// TIA Portal V21 export
DATA_BLOCK "ConfigDB"   // DB3
{ S7_Optimized_Access := 'TRUE' }
// stored: MemoryReserve 100
   VAR
      ksd1 : "coneCrusherConfigs";
   END_VAR
BEGIN
   ksd1.luS.self.timeToEstablishReturnFlow := T#60s;
   ksd1.luS.self.timeToEstablishFlow := T#15s;
   ksd1.luS.self.minOilFlow := 110.0;
   ksd1.luS.localModeSwitch.referenceDesignator := WSTRING#'LusLocalModeSw';
   ksd1.luS.localModeSwitch.onDelay := T#500ms;
   ksd1.luS.localModeSwitch.offDelay := T#200ms;
   ksd1.luS.btnStart.referenceDesignator := WSTRING#'LusBtnStart';
   ksd1.luS.btnStart.onDelay := T#500ms;
   ksd1.luS.btnStart.offDelay := T#200ms;
   ksd1.luS.btnStop.referenceDesignator := WSTRING#'LusBtnStop';
   ksd1.luS.btnStop.onDelay := T#500ms;
   ksd1.luS.btnStop.offDelay := T#200ms;
   ksd1.luS.btnReset.referenceDesignator := WSTRING#'LusBtnReset';
   ksd1.luS.btnReset.onDelay := T#500ms;
   ksd1.luS.btnReset.offDelay := T#200ms;
   ksd1.luS.oilPump1SelSwitch.referenceDesignator := WSTRING#'OilPump1Selected';
   ksd1.luS.oilPump1SelSwitch.onDelay := T#500ms;
   ksd1.luS.oilPump1SelSwitch.offDelay := T#200ms;
   ksd1.luS.oilPump2SelSwitch.referenceDesignator := WSTRING#'OilPump2Selected';
   ksd1.luS.oilPump2SelSwitch.onDelay := T#500ms;
   ksd1.luS.oilPump2SelSwitch.offDelay := T#200ms;
   ksd1.luS.oilPreparationSwitch.referenceDesignator := WSTRING#'OilPreparationSw';
   ksd1.luS.oilPreparationSwitch.onDelay := T#500ms;
   ksd1.luS.oilPreparationSwitch.offDelay := T#200ms;
   ksd1.luS.returnOilFlowSwitch.referenceDesignator := WSTRING#'ReturnOilFlowSw';
   ksd1.luS.returnOilFlowSwitch.onDelay := T#500ms;
   ksd1.luS.returnOilFlowSwitch.offDelay := T#200ms;
   ksd1.luS.oilLevelMax.referenceDesignator := WSTRING#'OilLevelMax';
   ksd1.luS.oilLevelMax.onDelay := T#500ms;
   ksd1.luS.oilLevelMax.offDelay := T#200ms;
   ksd1.luS.oilLevelMid.referenceDesignator := WSTRING#'OilLevelMid';
   ksd1.luS.oilLevelMid.onDelay := T#500ms;
   ksd1.luS.oilLevelMid.offDelay := T#200ms;
   ksd1.luS.oilLevelMin.referenceDesignator := WSTRING#'OilLevelMin';
   ksd1.luS.oilLevelMin.onDelay := T#500ms;
   ksd1.luS.oilLevelMin.offDelay := T#200ms;
   ksd1.luS.oilTempSwitchHigh.referenceDesignator := WSTRING#'OilTempSwHigh';
   ksd1.luS.oilTempSwitchHigh.onDelay := T#500ms;
   ksd1.luS.oilTempSwitchHigh.offDelay := T#200ms;
   ksd1.luS.oilTempSwitchLow.referenceDesignator := WSTRING#'OilTempSwLow';
   ksd1.luS.oilTempSwitchLow.onDelay := T#500ms;
   ksd1.luS.oilTempSwitchLow.offDelay := T#200ms;
   ksd1.luS.fbPump1.referenceDesignator := WSTRING#'FbPump1';
   ksd1.luS.fbPump1.onDelay := T#500ms;
   ksd1.luS.fbPump1.offDelay := T#200ms;
   ksd1.luS.fbPump2.referenceDesignator := WSTRING#'FbPump2';
   ksd1.luS.fbPump2.onDelay := T#500ms;
   ksd1.luS.fbPump2.offDelay := T#200ms;
   ksd1.luS.pump1Fault.referenceDesignator := WSTRING#'Pump1Fault';
   ksd1.luS.pump1Fault.onDelay := T#500ms;
   ksd1.luS.pump1Fault.offDelay := T#200ms;
   ksd1.luS.pump2Fault.referenceDesignator := WSTRING#'Pump2Fault';
   ksd1.luS.pump2Fault.onDelay := T#500ms;
   ksd1.luS.pump2Fault.offDelay := T#200ms;
   ksd1.luS.oilTempTank.referenceDesignator := WSTRING#'OilTempTank';
   ksd1.luS.oilTempTank.physicalUnit := 'C';
   ksd1.luS.oilTempTank.limitHigh2 := 60.0;
   ksd1.luS.oilTempTank.limitHigh1 := 55.0;
   ksd1.luS.oilTempTank.processValueMax := 120.0;
   ksd1.luS.oilTempTank.processValueMin := -50.0;
   ksd1.luS.oilTempTank.scaleAnalogUppPoint := 27648.0;
   ksd1.luS.oilTempTank.scaleProcessUppPoint := 120.0;
   ksd1.luS.oilTempTank.scaleProcessLowPoint := -50.0;
   ksd1.luS.oilPump1.referenceDesignator := WSTRING#'Pump1';
   ksd1.luS.oilPump1.startingControlTime := T#3s;
   ksd1.luS.oilPump1.stoppingControlTime := T#2s;
   ksd1.luS.oilPump1.disableFeedbackRunning := FALSE;
   ksd1.luS.oilPump1.disableFeedbackError := FALSE;
   ksd1.luS.oilPump2.referenceDesignator := WSTRING#'OilPump2';
   ksd1.luS.oilPump2.startingControlTime := T#3s;
   ksd1.luS.oilPump2.stoppingControlTime := T#2s;
   ksd1.luS.oilPump2.disableFeedbackRunning := FALSE;
   ksd1.luS.oilPump2.disableFeedbackError := FALSE;
   ksd1.luS.returnOilTemp.referenceDesignator := WSTRING#'ReturnOilTemp';
   ksd1.luS.returnOilTemp.physicalUnit := 'C';
   ksd1.luS.returnOilTemp.isUnipolarSignal := TRUE;
   ksd1.luS.returnOilTemp.limitHigh2 := 63.0;
   ksd1.luS.returnOilTemp.limitHigh1 := 60.0;
   ksd1.luS.returnOilTemp.processValueMax := 120.0;
   ksd1.luS.returnOilTemp.processValueMin := -50.0;
   ksd1.luS.returnOilTemp.scaleAnalogUppPoint := 27648.0;
   ksd1.luS.returnOilTemp.scaleAnalogLowPoint := 0.0;
   ksd1.luS.returnOilTemp.scaleProcessUppPoint := 120.0;
   ksd1.luS.returnOilTemp.scaleProcessLowPoint := -50.0;
   ksd1.luS.oilFlow.referenceDesignator := WSTRING#'OilFlow';
   ksd1.luS.oilFlow.physicalUnit := 'l/m';
   ksd1.luS.oilFlow.limitHigh2 := 500.0;
   ksd1.luS.oilFlow.limitHigh1 := 300.0;
   ksd1.luS.oilFlow.limitLow1 := 120.0;
   ksd1.luS.oilFlow.limitLow2 := 110.0;
   ksd1.luS.oilFlow.processValueMax := 300.0;
   ksd1.luS.oilFlow.processValueMin := 0.0;
   ksd1.luS.oilFlow.scaleAnalogUppPoint := 27648.0;
   ksd1.luS.oilFlow.scaleProcessUppPoint := 300.0;
   ksd1.luS.oilFlow.scaleProcessLowPoint := 0.0;
   ksd1.luS.inletWaterTemperature.referenceDesignator := WSTRING#'InletWaterTemp';
   ksd1.luS.inletWaterTemperature.physicalUnit := 'C';
   ksd1.luS.inletWaterTemperature.processValueMax := 120.0;
   ksd1.luS.inletWaterTemperature.processValueMin := -50.0;
   ksd1.luS.inletWaterTemperature.scaleAnalogUppPoint := 27648.0;
   ksd1.luS.inletWaterTemperature.scaleProcessUppPoint := 120.0;
   ksd1.luS.inletWaterTemperature.scaleProcessLowPoint := -50.0;
   ksd1.luS.outletWaterTemperature.referenceDesignator := WSTRING#'OutletWatertemp';
   ksd1.luS.outletWaterTemperature.physicalUnit := 'C';
   ksd1.luS.outletWaterTemperature.processValueMax := 120.0;
   ksd1.luS.outletWaterTemperature.processValueMin := -50.0;
   ksd1.luS.outletWaterTemperature.scaleAnalogUppPoint := 27648.0;
   ksd1.luS.outletWaterTemperature.scaleProcessUppPoint := 120.0;
   ksd1.luS.outletWaterTemperature.scaleProcessLowPoint := -50.0;
   ksd1.luS.inletOilTemperature.referenceDesignator := WSTRING#'InletOilTemp';
   ksd1.luS.inletOilTemperature.physicalUnit := 'C';
   ksd1.luS.inletOilTemperature.processValueMax := 120.0;
   ksd1.luS.inletOilTemperature.processValueMin := -50.0;
   ksd1.luS.inletOilTemperature.scaleAnalogUppPoint := 27648.0;
   ksd1.luS.inletOilTemperature.scaleAnalogLowPoint := 0.0;
   ksd1.luS.inletOilTemperature.scaleProcessUppPoint := 120.0;
   ksd1.luS.inletOilTemperature.scaleProcessLowPoint := -50.0;
   ksd1.luS.inletOilPressure.referenceDesignator := WSTRING#'InletOilPressure';
   ksd1.luS.inletOilPressure.physicalUnit := 'bar';
   ksd1.luS.inletOilPressure.processValueMax := 16.0;
   ksd1.luS.inletOilPressure.processValueMin := 0.0;
   ksd1.luS.inletOilPressure.scaleAnalogUppPoint := 27648.0;
   ksd1.luS.inletOilPressure.scaleAnalogLowPoint := 0.0;
   ksd1.luS.inletOilPressure.scaleProcessUppPoint := 16.0;
   ksd1.luS.inletOilPressure.scaleProcessLowPoint := 0.0;
   ksd1.luS.pump1Start.referenceDesignator := WSTRING#'Pump1Start';
   ksd1.luS.pump2Start.referenceDesignator := WSTRING#'Pump2Start';
   ksd1.luS.heaterOn.referenceDesignator := WSTRING#'HeaterOn';
   ksd1.luS.waterVlvOpen.referenceDesignator := WSTRING#'WaterVlvOpen';
   ksd1.luS.oilToCoolerVlv.referenceDesignator := WSTRING#'OilToCoolerVlv';
   ksd1.btnStart.referenceDesignator := WSTRING#'CrusherBtnStart';
   ksd1.btnStart.onDelay := T#500ms;
   ksd1.btnStart.offDelay := T#200ms;
   ksd1.btnStop.referenceDesignator := WSTRING#'CrusherBtnStop';
   ksd1.btnStop.onDelay := T#500ms;
   ksd1.btnStop.offDelay := T#200ms;
   ksd1.keySwitch.referenceDesignator := WSTRING#'CrusherKeySwitch';
   ksd1.keySwitch.onDelay := T#500ms;
   ksd1.emStop.referenceDesignator := WSTRING#'EmergencyStop';
   ksd1.emStop.onDelay := T#500ms;
   ksd1.btnReset.referenceDesignator := WSTRING#'CrusherBtnReset';
   ksd1.btnReset.onDelay := T#500ms;
   ksd1.btnReset.offDelay := T#200ms;
   ksd1.btnStartLuS.referenceDesignator := WSTRING#'CrusherBtnStartLus';
   ksd1.btnStartLuS.onDelay := T#500ms;
   ksd1.btnStartLuS.offDelay := T#200ms;
   ksd1.btnStopLuS.referenceDesignator := WSTRING#'CrusherBtnStopLus';
   ksd1.btnStopLuS.onDelay := T#500ms;
   ksd1.btnStopLuS.offDelay := T#200ms;
   ksd1.premoldingSw.referenceDesignator := WSTRING#'PremoldingSw';
   ksd1.premoldingSw.onDelay := T#500ms;
   ksd1.premoldingSw.offDelay := T#500ms;
   ksd1.crusherEccentricTemp.referenceDesignator := WSTRING#'EccentricTemp';
   ksd1.crusherEccentricTemp.physicalUnit := 'C';
   ksd1.crusherEccentricTemp.isUnipolarSignal := TRUE;
   ksd1.crusherEccentricTemp.limitHigh2 := 70.0;
   ksd1.crusherEccentricTemp.limitHigh1 := 60.0;
   ksd1.crusherEccentricTemp.processValueMax := 120.0;
   ksd1.crusherEccentricTemp.processValueMin := -50.0;
   ksd1.crusherEccentricTemp.scaleAnalogUppPoint := 27648.0;
   ksd1.crusherEccentricTemp.scaleAnalogLowPoint := 0.0;
   ksd1.crusherEccentricTemp.scaleProcessUppPoint := 120.0;
   ksd1.crusherEccentricTemp.scaleProcessLowPoint := -50.0;
   ksd1.crusherOuterBearingTemp.referenceDesignator := WSTRING#'CrusherOuterBearTemp';
   ksd1.crusherOuterBearingTemp.physicalUnit := 'C';
   ksd1.crusherOuterBearingTemp.isUnipolarSignal := TRUE;
   ksd1.crusherOuterBearingTemp.limitHigh2 := 70.0;
   ksd1.crusherOuterBearingTemp.limitHigh1 := 60.0;
   ksd1.crusherOuterBearingTemp.processValueMax := 120.0;
   ksd1.crusherOuterBearingTemp.processValueMin := -50.0;
   ksd1.crusherOuterBearingTemp.scaleAnalogUppPoint := 27648.0;
   ksd1.crusherOuterBearingTemp.scaleAnalogLowPoint := 0.0;
   ksd1.crusherOuterBearingTemp.scaleProcessUppPoint := 120.0;
   ksd1.crusherOuterBearingTemp.scaleProcessLowPoint := -50.0;
   ksd1.crusherInnerBearingTemp.referenceDesignator := WSTRING#'CrusherInnerBearTemp';
   ksd1.crusherInnerBearingTemp.physicalUnit := 'C';
   ksd1.crusherInnerBearingTemp.isUnipolarSignal := TRUE;
   ksd1.crusherInnerBearingTemp.limitHigh2 := 70.0;
   ksd1.crusherInnerBearingTemp.limitHigh1 := 60.0;
   ksd1.crusherInnerBearingTemp.processValueMax := 120.0;
   ksd1.crusherInnerBearingTemp.processValueMin := -50.0;
   ksd1.crusherInnerBearingTemp.scaleAnalogUppPoint := 27648.0;
   ksd1.crusherInnerBearingTemp.scaleAnalogLowPoint := 0.0;
   ksd1.crusherInnerBearingTemp.scaleProcessUppPoint := 120.0;
   ksd1.crusherInnerBearingTemp.scaleProcessLowPoint := -50.0;
   ksd1.driveFrontBearingTemp.referenceDesignator := WSTRING#'DriveFrontBearTemp';
   ksd1.driveFrontBearingTemp.physicalUnit := 'C';
   ksd1.driveFrontBearingTemp.isUnipolarSignal := TRUE;
   ksd1.driveFrontBearingTemp.limitHigh2 := 70.0;
   ksd1.driveFrontBearingTemp.limitHigh1 := 60.0;
   ksd1.driveFrontBearingTemp.processValueMax := 120.0;
   ksd1.driveFrontBearingTemp.processValueMin := -50.0;
   ksd1.driveFrontBearingTemp.scaleAnalogUppPoint := 27648.0;
   ksd1.driveFrontBearingTemp.scaleAnalogLowPoint := 0.0;
   ksd1.driveFrontBearingTemp.scaleProcessUppPoint := 120.0;
   ksd1.driveFrontBearingTemp.scaleProcessLowPoint := -50.0;
   ksd1.driveRearBearingTemp.referenceDesignator := WSTRING#'DriveRearBearTemp';
   ksd1.driveRearBearingTemp.physicalUnit := 'C';
   ksd1.driveRearBearingTemp.isUnipolarSignal := TRUE;
   ksd1.driveRearBearingTemp.limitHigh2 := 70.0;
   ksd1.driveRearBearingTemp.limitHigh1 := 60.0;
   ksd1.driveRearBearingTemp.processValueMax := 120.0;
   ksd1.driveRearBearingTemp.processValueMin := -50.0;
   ksd1.driveRearBearingTemp.scaleAnalogUppPoint := 27648.0;
   ksd1.driveRearBearingTemp.scaleAnalogLowPoint := 0.0;
   ksd1.driveRearBearingTemp.scaleProcessUppPoint := 120.0;
   ksd1.driveRearBearingTemp.scaleProcessLowPoint := -50.0;
   ksd1.driveWindingTempP1.referenceDesignator := WSTRING#'DriveWindingTempP1';
   ksd1.driveWindingTempP1.physicalUnit := 'C';
   ksd1.driveWindingTempP1.isUnipolarSignal := TRUE;
   ksd1.driveWindingTempP1.default := 0.0;
   ksd1.driveWindingTempP1.limitHigh2 := 80.0;
   ksd1.driveWindingTempP1.limitHigh1 := 70.0;
   ksd1.driveWindingTempP1.limitLow1 := -200.0;
   ksd1.driveWindingTempP1.limitLow2 := -270.0;
   ksd1.driveWindingTempP1.processValueMax := 120.0;
   ksd1.driveWindingTempP1.processValueMin := -50.0;
   ksd1.driveWindingTempP1.scaleAnalogUppPoint := 27648.0;
   ksd1.driveWindingTempP1.scaleAnalogLowPoint := 0.0;
   ksd1.driveWindingTempP1.scaleProcessUppPoint := 120.0;
   ksd1.driveWindingTempP1.scaleProcessLowPoint := -50.0;
   ksd1.driveWindingTempP1.disableAlarms := FALSE;
   ksd1.driveWindingTempP2.referenceDesignator := WSTRING#'DriveWindingTempP2';
   ksd1.driveWindingTempP2.physicalUnit := 'C';
   ksd1.driveWindingTempP2.isUnipolarSignal := TRUE;
   ksd1.driveWindingTempP2.default := 0.0;
   ksd1.driveWindingTempP2.limitHigh2 := 80.0;
   ksd1.driveWindingTempP2.limitHigh1 := 70.0;
   ksd1.driveWindingTempP2.limitLow1 := -200.0;
   ksd1.driveWindingTempP2.limitLow2 := -270.0;
   ksd1.driveWindingTempP2.processValueMax := 120.0;
   ksd1.driveWindingTempP2.processValueMin := -50.0;
   ksd1.driveWindingTempP2.scaleAnalogUppPoint := 27648.0;
   ksd1.driveWindingTempP2.scaleAnalogLowPoint := 0.0;
   ksd1.driveWindingTempP2.scaleProcessUppPoint := 120.0;
   ksd1.driveWindingTempP2.scaleProcessLowPoint := -50.0;
   ksd1.driveWindingTempP2.disableAlarms := FALSE;
   ksd1.driveWindingTempP3.referenceDesignator := WSTRING#'DriveWindingTempP3';
   ksd1.driveWindingTempP3.physicalUnit := 'C';
   ksd1.driveWindingTempP3.isUnipolarSignal := TRUE;
   ksd1.driveWindingTempP3.default := 0.0;
   ksd1.driveWindingTempP3.limitHigh2 := 80.0;
   ksd1.driveWindingTempP3.limitHigh1 := 70.0;
   ksd1.driveWindingTempP3.limitLow1 := -200.0;
   ksd1.driveWindingTempP3.limitLow2 := -270.0;
   ksd1.driveWindingTempP3.processValueMax := 120.0;
   ksd1.driveWindingTempP3.processValueMin := -50.0;
   ksd1.driveWindingTempP3.scaleAnalogUppPoint := 27648.0;
   ksd1.driveWindingTempP3.scaleAnalogLowPoint := 0.0;
   ksd1.driveWindingTempP3.scaleProcessUppPoint := 120.0;
   ksd1.driveWindingTempP3.scaleProcessLowPoint := -50.0;
   ksd1.driveWindingTempP3.disableAlarms := FALSE;
   ksd1.driveCurrent.referenceDesignator := WSTRING#'DriveCurrent';
   ksd1.driveCurrent.physicalUnit := 'A';
   ksd1.driveCurrent.isUnipolarSignal := TRUE;
   ksd1.driveCurrent.default := 0.0;
   ksd1.driveCurrent.limitHigh2 := 100.0;
   ksd1.driveCurrent.limitHigh1 := 80.0;
   ksd1.driveCurrent.limitLow1 := -200.0;
   ksd1.driveCurrent.limitLow2 := -270.0;
   ksd1.driveCurrent.processValueMax := 200.0;
   ksd1.driveCurrent.processValueMin := 0.0;
   ksd1.driveCurrent.scaleAnalogUppPoint := 27648.0;
   ksd1.driveCurrent.scaleAnalogLowPoint := 0.0;
   ksd1.driveCurrent.scaleProcessUppPoint := 200.0;
   ksd1.driveCurrent.scaleProcessLowPoint := 0.0;
   ksd1.driveCurrent.disableAlarms := FALSE;
   ksd1.sgReady.referenceDesignator := WSTRING#'SgReady';
   ksd1.sgReady.onDelay := T#500ms;
   ksd1.sgReady.offDelay := T#500ms;
   ksd1.sgReady.invertProcessValue := FALSE;
   ksd1.sgFbOn.referenceDesignator := WSTRING#'SgFbOn';
   ksd1.sgFbOn.onDelay := T#500ms;
   ksd1.sgFbOn.offDelay := T#500ms;
   ksd1.sgFbOff.referenceDesignator := WSTRING#'SgFbOff';
   ksd1.sgFbOff.onDelay := T#500ms;
   ksd1.sgFbOff.offDelay := T#500ms;
   ksd1.sgStart.referenceDesignator := WSTRING#'SwitchgearStart';
   ksd1.sgStart.default := FALSE;
   ksd1.sgStart.invertProcessValue := FALSE;
   ksd1.sgStart.disableAlarms := FALSE;
   ksd1.sgStop.referenceDesignator := WSTRING#'SwitchgearStop';
   ksd1.sgStop.default := TRUE;
   ksd1.sgStop.invertProcessValue := FALSE;
   ksd1.sgStop.disableAlarms := FALSE;
   ksd1.preStartAlmOn.referenceDesignator := WSTRING#'PreStartAlmOn';
   ksd1.preStartAlmOn.default := FALSE;
   ksd1.preStartAlmOn.invertProcessValue := FALSE;
   ksd1.preStartAlmOn.disableAlarms := FALSE;
   ksd1.feedEn.referenceDesignator := WSTRING#'FeedEn';
   ksd1.feedEn.default := FALSE;
   ksd1.feedEn.invertProcessValue := FALSE;
   ksd1.feedEn.disableAlarms := FALSE;
   ksd1.preStartAlmFb.referenceDesignator := WSTRING#'PreStartAlmFb';
   ksd1.preStartAlmFb.onDelay := T#500ms;
   ksd1.preStartAlmFb.offDelay := T#500ms;
   ksd1.preStartAlmFb.default := FALSE;
   ksd1.preStartAlmFb.invertProcessValue := FALSE;
   ksd1.preStartAlmFb.disableAlarms := FALSE;
END_DATA_BLOCK
